RoboDK station: Simulation.rdk

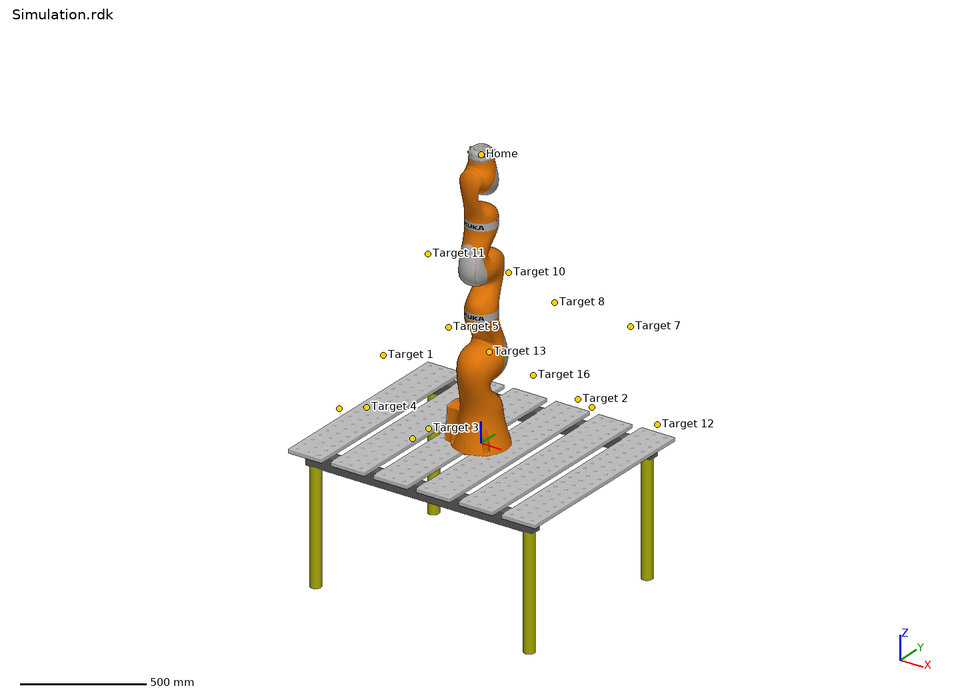
[picture v0: the station drawn from its stored meshes, robots at their saved joint values, targets as dots, program paths as lines]
Station Simulation. Poses are relative to the parent item; angles as X-Y-Z fixed-axis rotations.
Station parameters (name, value as stored): CollisionFreePlanner, KUKA LBR iiwa 14 R820, CollisionFreePlanner-Rob KUKA LBR iiwa 14 R820
  - frame KUKA LBR iiwa 14 R820 Base at (0, 1000, 0) mm
    - robot KUKA LBR iiwa 14 R820: 7 axes, payload 14 kg, reach 1180 mm, repeatability 0.15 mm, weight 29.9 kg
        modified DH rows (alpha deg, a mm, theta deg, d mm): 0, 0, 0, 360; -90, 0, 0, 0; 90, 0, 0, 420; -90, 0, 0, 0; 90, 0, 0, 400; -90, 0, 0, 0; 90, 0, 0, 90
        joint limits [-170, -120, -170, -120, -170, -120, -175] to [170, 120, 170, 120, 170, 120, 175]; home [0, 0, 0, -90, 0, 0, 0]; saved at [0, 0, 0, 0, 0, 0, 0]
    - object Object Table at (0, 0, 0) mm, size 1193.8 x 965.2 x 609.6 mm, geometry from Object Table.wrl
    - target Target 1 (joint target) at (-315.2, -225.57, 388.93) mm, rotated rx 71.23 ry -2.75 rz 112.11 deg; joints [-20, -90, -90, -110, -160, -110, -170] of KUKA LBR iiwa 14 R820
    - target Target 2 (joint target) at (543.75, -107.65, 388.93) mm, rotated rx -70.45 ry 16.16 rz -85.53 deg; joints [40, 90, -90, -110, -160, 70, -170] of KUKA LBR iiwa 14 R820
    - target Target 3 (joint target) at (212.97, -665.2, 388.93) mm, rotated rx 71.23 ry -2.75 rz 87.11 deg; joints [135, -90, -90, 70, -160, -110, -170] of KUKA LBR iiwa 14 R820
    - target Target 4 (joint target) at (-99.72, -647.59, 388.93) mm, rotated rx -70.45 ry 16.16 rz -85.53 deg; joints [-140, 90, -90, 70, -160, 70, -170] of KUKA LBR iiwa 14 R820
    - target Target 5 (joint target) at (-315.2, 225.57, 331.07) mm, rotated rx 108.77 ry -2.75 rz 67.89 deg; joints [20, -90, 90, -110, -160, -110, 10] of KUKA LBR iiwa 14 R820
    - target Target 6 (joint target) at (551.07, 59.85, 331.07) mm, rotated rx -109.55 ry 16.16 rz -99.47 deg; joints [-45, 90, 90, -110, -160, 70, 10] of KUKA LBR iiwa 14 R820
    - target Target 7 (joint target) at (270.14, 644.1, 331.07) mm, rotated rx 108.77 ry -2.75 rz 87.89 deg; joints [-140, -90, 90, 70, -160, -110, 10] of KUKA LBR iiwa 14 R820
    - target Target 8 (joint target) at (-99.72, 647.59, 331.07) mm, rotated rx -109.55 ry 16.16 rz -94.47 deg; joints [140, 90, 90, 70, -160, 70, 10] of KUKA LBR iiwa 14 R820
    - target Target 9 (joint target) at (286.48, 354.23, 97.35) mm, rotated rx -103.52 ry 1.49 rz -88.52 deg; joints [-165, -90, -130, -110, 20, -110, -130] of KUKA LBR iiwa 14 R820
    - target Target 10 (joint target) at (-111.56, 348.62, 580.57) mm, rotated rx -148.51 ry -74.09 rz -34.33 deg; joints [165, 90, -130, -110, 20, 70, -130] of KUKA LBR iiwa 14 R820
    - target Target 11 (joint target) at (-471.6, 305.2, 578.33) mm, rotated rx -160.67 ry 74.09 rz -148.51 deg; joints [0, -90, -130, 70, 20, -110, -130] of KUKA LBR iiwa 14 R820
    - target Target 12 (joint target) at (585.26, 378.05, 95.11) mm, rotated rx 105.52 ry -14.86 rz 84.48 deg; joints [10, 90, -130, 70, 20, 70, -130] of KUKA LBR iiwa 14 R820
    - target Target 13 (joint target) at (286.48, -354.23, 622.65) mm, rotated rx -76.48 ry 1.49 rz -91.48 deg; joints [165, -90, 50, -110, 20, -110, 50] of KUKA LBR iiwa 14 R820
    - target Target 14 (joint target) at (-80.75, -357.02, 139.43) mm, rotated rx -31.49 ry -74.09 rz -140.67 deg; joints [-160, 90, 50, -110, 20, 70, 50] of KUKA LBR iiwa 14 R820
    - target Target 15 (joint target) at (-471.6, -305.2, 141.67) mm, rotated rx -19.33 ry 74.09 rz -31.49 deg; joints [0, -90, 50, 70, 20, -110, 50] of KUKA LBR iiwa 14 R820
    - target Target 16 (joint target) at (550.08, -427.62, 624.89) mm, rotated rx 74.48 ry -14.86 rz 90.52 deg; joints [-15, 90, 50, 70, 20, 70, 50] of KUKA LBR iiwa 14 R820
    - target Home (joint target) at (0, 0, 1270) mm; joints [0, 0, 0, 0, 0, 0, 0] of KUKA LBR iiwa 14 R820
